(* PLC project Unnamed, Unknown Unnamed 1 *)
(* stored: creationDateTime 2023-03-06T07:03:38, modificationDateTime 2023-03-19T23:08:22 *)

PROGRAM SWITCHVSLAMPS
  VAR_INPUT
    PB1 : BOOL;  (* TURNS ON:L1,L2,L3 *)
    PB2 : BOOL;  (* TURNS ON:L4,L5,L6 *)
    PB3 : BOOL;  (* TURNS ON:L7,L8,L9 *)
    PB4 : BOOL;  (* TURNS OFF:L1,L5,L9 *)
    PB5 : BOOL;  (* TURNS OFF:L3,L4,L8 *)
    PB6 : BOOL;  (* TURNS OFF:L2,L6,L7 *)
    PB7 : BOOL;  (* TURNS OFF ALL LAMPS *)
  END_VAR
  VAR_OUTPUT
    L1 : BOOL;
    L2 : BOOL;
    L3 : BOOL;
    L4 : BOOL;
    L5 : BOOL;
    L6 : BOOL;
    L7 : BOOL;
    L8 : BOOL;
    L9 : BOOL;
  END_VAR
  VAR
    SR0 : SR;
    SR1 : SR;
    SR2 : SR;
    SR3 : SR;
    SR4 : SR;
    SR5 : SR;
    SR6 : SR;
    SR7 : SR;
    SR8 : SR;
  END_VAR

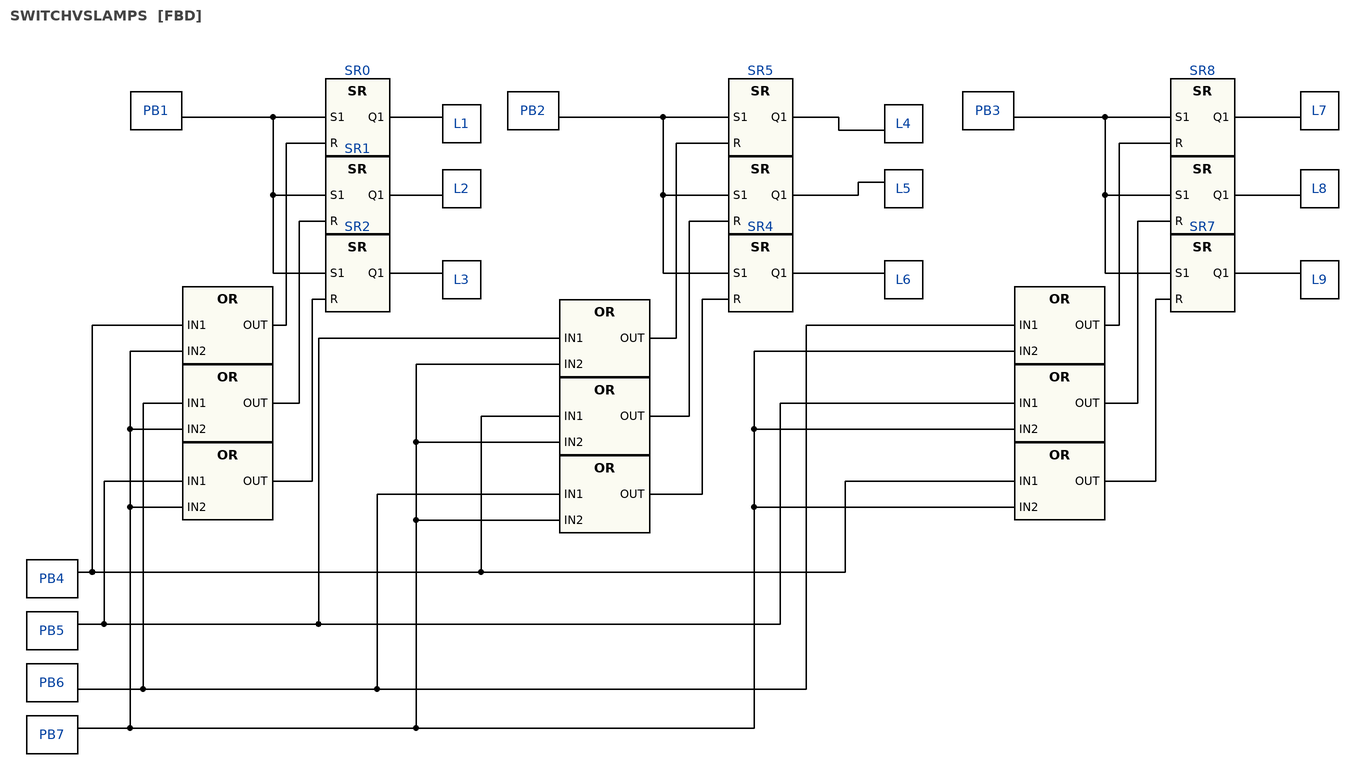
(* FBD diagram, written out as Structured Text *)
SR8(S1 := PB3, R := PB6 OR PB7);
L7 := SR8.Q1;
SR0(S1 := PB1, R := PB4 OR PB7);
L1 := SR0.Q1;
SR5(S1 := PB2, R := PB5 OR PB7);
L4 := SR5.Q1;
SR1(S1 := PB1, R := PB6 OR PB7);
L2 := SR1.Q1;
SR3(S1 := PB2, R := PB4 OR PB7);
L5 := SR3.Q1;
SR6(S1 := PB3, R := PB5 OR PB7);
L8 := SR6.Q1;
SR2(S1 := PB1, R := PB5 OR PB7);
L3 := SR2.Q1;
SR4(S1 := PB2, R := PB6 OR PB7);
L6 := SR4.Q1;
SR7(S1 := PB3, R := PB4 OR PB7);
L9 := SR7.Q1;
END_PROGRAM

CONFIGURATION Config0
  RESOURCE Res0 ON PLC
    TASK task0(INTERVAL := T#20ms, PRIORITY := 0);
    PROGRAM instance0 WITH task0 : SWITCHVSLAMPS;
  END_RESOURCE
END_CONFIGURATION
